FUNCTION_BLOCK FB_ExampleDeviceSM
VAR_INPUT
END_VAR
VAR_OUTPUT
	fReqAtt	:	REAL;
END_VAR
VAR
END_VAR

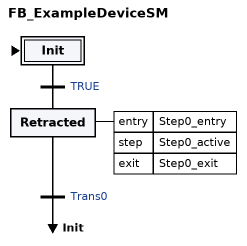
INITIAL_STEP Init:
END_STEP
TRANSITION FROM Init TO Retracted
    := TRUE;
END_TRANSITION
STEP Retracted:
    Step0_entry(P1);  // entry action
    Step0_active(N);  // step action
    Step0_exit(P0);  // exit action
END_STEP
TRANSITION FROM Retracted TO Init
    := Trans0;
END_TRANSITION

ACTION Step0_active:

END_ACTION

ACTION Step0_entry:

END_ACTION

ACTION Step0_exit:

END_ACTION

END_FUNCTION_BLOCK

(* stored: Version 1.1.0.1, ProductVersion 3.1.4022.10
   POU FB_ExampleDeviceSM: Id {add7e2f6-5264-48b5-8412-2ce66fdaf036}, SpecialFunc None
   Action Step0_active: Id {0d71acd4-38e2-4ca6-bfe8-4a38cbcd4923}
   Action Step0_entry: Id {f127fba7-ea8c-4224-a26b-fbb04a9e74d7}
   Action Step0_exit: Id {07f8f338-67e6-4912-be8e-f5961f122162} *)
